TYPE Location :
STRUCT
	Piece: Piece;
	Done: BOOL := FALSE;
	Occupied: BOOL := FALSE;
	Processed: BOOL := FALSE;
END_STRUCT
END_TYPE

(* stored: Version 1.1.0.1, ProductVersion 3.1.4024.12
   DUT Location: Id {293857e0-8485-4910-9271-377f3b56bd4c} *)
